PROGRAM MobjectDisposableUnitTests
VAR
	disposable_TestSuite : Disposable_TestSuite;
END_VAR

END_PROGRAM

(* stored: Version 1.1.0.1, ProductVersion 3.1.4024.12
   POU MobjectDisposableUnitTests: Id {16004530-efeb-0415-1922-33cae33576f7}, SpecialFunc None *)
